{attribute 'qualified_only'}
{attribute 'to_string'}
TYPE E_DataBaseTable :
(
	NoError := 0,
	HardwareConfig_ReadFail,
	HardwareConfig_ReadDataOutOfRange,
	HardwareConfig_InputReferenceInvaild,
	HardwareConfig_NoData,
	MachineParameter_ReadFail,
	MachineParameter_ReadDataOutOfRange,
	MachineParameter_InputReferenceInvaild,
	MachineParameter_NoData,
	MachineParameter_FillDataToSubsysFail,
	MachineParameter_FillDataToCoreSysFail,
	MachineParameter_FillDataToMachineFail,
	MessageList_ReadFail,
	MessageList_ReadDataOutOfRange,	
	MessageList_InputReferenceInvaild,
	MessageList_NoData,
	MessageList_MessageCodeOrArraySizeOutOfRange,
	AlarmHistory_UploadDataFail,
	DataUpload_ConnectToDBFail,
	DataUpload_AlarmHistoryBufferFull,
	DataUpload_AlarmHistoryUploadFail,
	DataUpload_AlarmHistoryUploadFailWriteDataToFileFail, //重大異常，不能直接reset需要人員排查原因，程式內部鎖死不能reset
	DataUpload_ProductionHistoryBufferFull,
	DataUpload_ProductionHistoryUploadFail,
	DataUpload_ProductionHistoryWriteDataToFileFail, //重大異常，不能直接reset需要人員排查原因，程式內部鎖死不能reset
	DataUpload_ProductionReportBufferFull,
	DataUpload_ProductionReportUploadFail,
	DataUpload_ProductionReportWriteDataToFileFail, //重大異常，不能直接reset需要人員排查原因，程式內部鎖死不能reset
	DataUpload_ProductionSummaryBufferFull,
	DataUpload_ProductionSummaryUploadFail,
	DataUpload_ProductionSummaryWriteDataToFileFail, //重大異常，不能直接reset需要人員排查原因，程式內部鎖死不能reset
	DataUpload_SoDurationBufferFull,
	DataUpload_SoDurationUploadFail,
	DataUpload_SoDurationWriteDataToFileFail, //重大異常，不能直接reset需要人員排查原因，程式內部鎖死不能reset
	DataUpload_StopCountBufferFull,	
	DataUpload_StopCountUploadFail,
	DataUpload_StopCountWriteDataToFileFail, //重大異常，不能直接reset需要人員排查原因，程式內部鎖死不能reset
	DataUpload_RegularCheckResultsBufferFull,
	DataUpload_RegularCheckResultsUploadFail,
	DataUpload_RegularCheckResultsWriteDataToFileFail, //重大異常，不能直接reset需要人員排查原因，程式內部鎖死不能reset
	ProductionReport_UploadDataFail,
	ProductionSummary_UploadDataFail,
	ProductionHistoryInspection_UploadDataFail,
	RegularCheckResults_UploadDataFail,
	SoDuration_UploadDataFail,
	StopCount_UploadDataFail,
	CheckDBconnection_ReadDBStatusTimeout,
	CheckDBconnection_RetryConnectToDBFail,
	CheckDBconnection_StatusDataOutOfRange,
	ProdHistoryProcedure_UploadDataFail,
	ProdHistoryProcedure_WriteDataToFileFail, //重大異常，不能直接reset需要人員排查原因，程式內部鎖死不能reset
	ProdHistoryProcedure_InputInterfaceInvalid,
	ProdStatusChangedStopCount_FillDataTimeout,
	ProdStatusChangedStopCount_AddDataToBufferTimeout,
	UploadEndBatchData_FillProductionReportDataTimeout,
	UploadEndBatchData_FillProductionSummaryDataTimeout,
	UploadEndBatchData_FillSoDurationDataTimeout,
	UploadEndBatchData_AddProductionReportDataToBufferTimeout,
	UploadEndBatchData_AddProductionSummaryDataToBufferTimeout,
	UploadEndBatchData_AddSoDurationDataToBufferTimeout,
	UploadProdRegularReport_FillProductionReportDataTimeout,
	UploadProdRegularReport_AddProductionReportDataToBufferTimeout
	
	
)UDINT;
END_TYPE

(* stored: Version 1.1.0.1, ProductVersion 3.1.4024.11
   EnumerationTextList E_DataBaseTable: Id {65fcec10-34f7-4819-8a93-df39bd6ffc18} *)
